// TIA Portal project "ProjetoCLP-TiaPortal" (V16)

(* hardware
DEVICE "S71500/ET200MP station_1"  S7-1500 station
   slot 0: "Rail_0"  Rack  6ES7 590-1***0-0AA0
   slot 1: "PLC_1"  CPU 1511-1 PN  6ES7 511-1AK01-0AB0  V2.8
      slot 3: "CPU display_1"  6ES7591-1AA00-0AA0
      slot 32768: "PROFINET interface_1"  X1
         slot 32769: "Port_1"  X1 P1
         slot 32770: "Port_2"  X1 P2
      slot 34817: "Virtual CP interface port_1"  Virtual CP interface port  Virtual CP interface port
*)

// ===== PLC "PLC_1"  CPU 1511-1 PN =====

VAR_GLOBAL   // PLC tag table "Default tag table"
   "TemperaturaEntrada" AT %ID112 : Real;
   "SaidaTemperatura" AT %QW112 : Int;
   "Display" AT %QD100 : Real;
   "Stop" AT %I0.0 : Bool;
   "Motor 1" AT %Q0.0 : Bool;
   "Start" AT %I0.1 : Bool;
   "Tag_2" AT %Q0.5 : Bool;
   "Tag_3" AT %Q0.4 : Bool;
   "Tag_4" AT %Q0.3 : Bool;
   "Tag_5" AT %Q0.2 : Bool;
   "Tag_6" AT %Q0.1 : Bool;
   "IsOn" AT %Q0.6 : Bool;
END_VAR

DATA_BLOCK "Entrada analogica"   // DB1
{ S7_Optimized_Access := 'TRUE' }
VERSION : 0.1
   VAR
      tempAnalogico : Real := 0.0;
   END_VAR
BEGIN
END_DATA_BLOCK

ORGANIZATION_BLOCK "Main"   // OB1, LAD, ProgramCycle
TITLE = "Main Program Sweep (Cycle)"
{ S7_Optimized_Access := 'TRUE' }
VERSION : 0.1
   VAR_INPUT
      Initial_Call : Bool;   // Initial call of this OB
      Remanence : Bool;   // =True, if remanent data are available
   END_VAR
   VAR_TEMP
      norm : Real;
      norm2 : Real;
   END_VAR
BEGIN

REGION Network 1
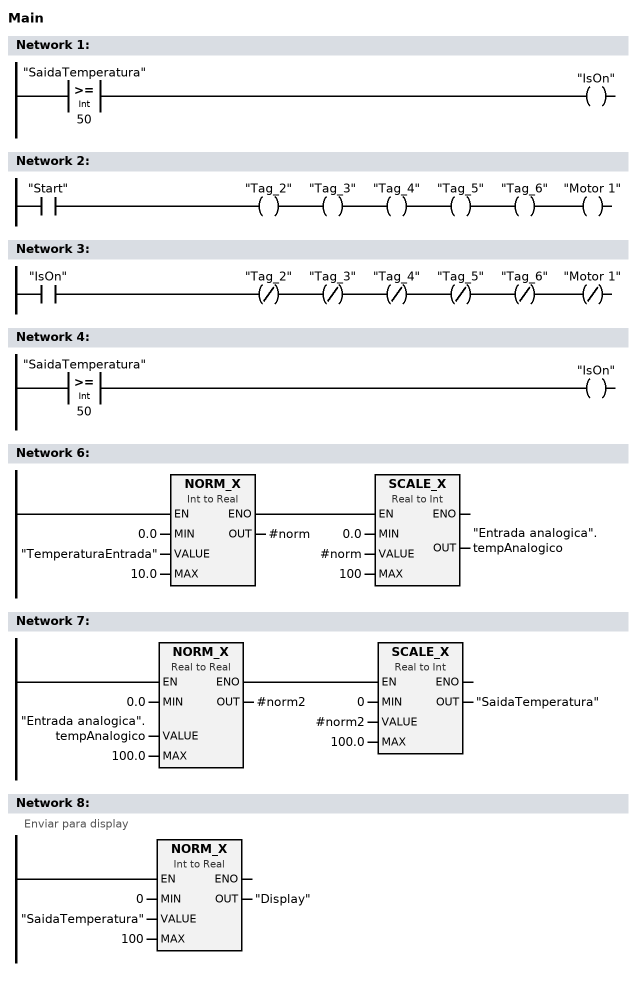
   RUNG wire#powerrail
      { S7_Templates := "SrcType := Int" } GE_Contact(in1 := "SaidaTemperatura", in2 := 50)
      Coil( "IsOn" )
   END_RUNG
   // the same network as SCL:
   "IsOn" := "SaidaTemperatura" >= 50;
END_REGION

REGION Network 2
   RUNG wire#powerrail
      Contact( "Start" )
      Coil( "Tag_2" )
      Coil( "Tag_3" )
      Coil( "Tag_4" )
      Coil( "Tag_5" )
      Coil( "Tag_6" )
      Coil( "Motor 1" )
   END_RUNG
   // the same network as SCL:
   "Tag_2" := "Start";
   "Tag_3" := "Start";
   "Tag_4" := "Start";
   "Tag_5" := "Start";
   "Tag_6" := "Start";
   "Motor 1" := "Start";
END_REGION

REGION Network 3
   RUNG wire#powerrail
      Contact( "IsOn" )
      I_Coil( "Tag_2" )
      I_Coil( "Tag_3" )
      I_Coil( "Tag_4" )
      I_Coil( "Tag_5" )
      I_Coil( "Tag_6" )
      I_Coil( "Motor 1" )
   END_RUNG
   // the same network as SCL:
   "Tag_2" := NOT "IsOn";
   "Tag_3" := NOT "IsOn";
   "Tag_4" := NOT "IsOn";
   "Tag_5" := NOT "IsOn";
   "Tag_6" := NOT "IsOn";
   "Motor 1" := NOT "IsOn";
END_REGION

REGION Network 4
   RUNG wire#powerrail
      { S7_Templates := "SrcType := Int" } GE_Contact(in1 := "SaidaTemperatura", in2 := 50)
      Coil( "IsOn" )
   END_RUNG
   // the same network as SCL:
   "IsOn" := "SaidaTemperatura" >= 50;
END_REGION

REGION Network 6
   RUNG wire#powerrail
      { S7_Templates := "[SrcType := Int, DestType := Real]" } Normalize(min := 0.0, value := "TemperaturaEntrada", max := 10.0, out => #norm)
      { S7_Templates := "[SrcType := Real, DestType := Int]" } Scale(min := 0.0, value := #norm, max := 100, out => "Entrada analogica".tempAnalogico)
   END_RUNG
   // the same network as SCL:
   #norm := NORM_X(MIN := 0.0, VALUE := "TemperaturaEntrada", MAX := 10.0);
   "Entrada analogica".tempAnalogico := SCALE_X(MIN := 0.0, VALUE := #norm, MAX := 100);
END_REGION

REGION Network 7
   RUNG wire#powerrail
      { S7_Templates := "[SrcType := Real, DestType := Real]" } Normalize(min := 0.0, value := "Entrada analogica".tempAnalogico, max := 100.0, out => #norm2)
      { S7_Templates := "[SrcType := Real, DestType := Int]" } Scale(min := 0, value := #norm2, max := 100.0, out => "SaidaTemperatura")
   END_RUNG
   // the same network as SCL:
   #norm2 := NORM_X(MIN := 0.0, VALUE := "Entrada analogica".tempAnalogico, MAX := 100.0);
   "SaidaTemperatura" := SCALE_X(MIN := 0, VALUE := #norm2, MAX := 100.0);
END_REGION

REGION Network 8
   // Enviar para display
   RUNG wire#powerrail
      { S7_Templates := "[SrcType := Int, DestType := Real]" } Normalize(min := 0, value := "SaidaTemperatura", max := 100, out => "Display")
   END_RUNG
   // the same network as SCL:
   "Display" := NORM_X(MIN := 0, VALUE := "SaidaTemperatura", MAX := 100);
END_REGION
END_ORGANIZATION_BLOCK